// TIA Portal V19 export
TYPE "LEXCHANGETRAY_typeCustomerAlarmInterface"
// stored: Access Published
   STRUCT
      error : "type_errorInterface";
   END_STRUCT;
END_TYPE
